// Mitsubishi GX Works2 project: Flip-flop practice 1   PLC: Q00J

PROGRAM MAIN
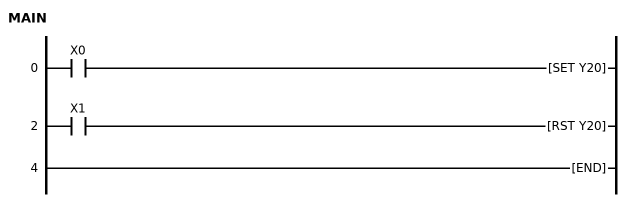
0     LD      X0
      SET     Y20
2     LD      X1
      RST     Y20
4     END
END_PROGRAM
